FUNCTION_BLOCK Signal EXTENDS InstancePath IMPLEMENTS IBaseSignal, IDifferentiable, ISignal
VAR
    _out : LREAL;
    _derivative : Derivative;
    _iir : InfiniteImpulseResponse;
    _controller : IController;
END_VAR

METHOD Control : IOut
VAR_INPUT
    setpoint : LREAL;
END_VAR
IF _controller <> 0 THEN
    _controller.Update(setpoint:=setpoint, actual:=THIS^.Out);
    _out := _controller.Out;
    Control := THIS^;
ELSE
    ADSLOGSTR(
        msgCtrlMask:=ADSLOG_MSGTYPE_ERROR,
        msgFmtStr:='%s: Assign a controller before calling this method.',
        strArg:=_path
    );
END_IF
END_METHOD

PROPERTY Controller : IController
SET
_controller := Controller;
END_SET
END_PROPERTY

METHOD Differentiate : IDifferentiable
VAR_INPUT
    deltaTime : Millisecond;
END_VAR
_derivative(value:=THIS^.Out, deltaTime:=deltaTime);
_out := _derivative.Out;
Differentiate := THIS^;
END_METHOD

METHOD Iir : IBaseSignal
VAR_INPUT
    decay : LREAL;
END_VAR
_iir(new:=THIS^.Out, decay:=decay);
_out := _iir.Out;
Iir := THIS^;
END_METHOD

PROPERTY Out : LREAL
GET
OUT := _out;
END_GET
END_PROPERTY

METHOD Update : ISignal
VAR_INPUT
    value : LREAL;
END_VAR
_out := value;
Update := THIS^;
END_METHOD

END_FUNCTION_BLOCK

(* stored: Version 1.1.0.1
   POU Signal: Id {d5e65a98-c59a-40a4-8e08-14b2a0104701}, SpecialFunc None
   Method Control: Id {8dcf8e28-9ea3-49a8-b60f-0e1e6205b9e1}
   Property Controller: Id {7fb07e13-2348-48d3-8313-9eff675207f8}
   Set Set: Id {17a680e5-7bae-43e2-91a2-a31ebdb6de08}
   Method Differentiate: Id {3cb626dd-f306-4dd7-8b41-c5d14146e141}
   Method Iir: Id {20733bae-2f54-4e93-a73e-666694dd4f84}
   Property Out: Id {f11c0c9d-cbae-4516-9e11-e42329123126}
   Get Get: Id {42b506ae-6bce-45b3-bdd7-aeb51ebf09f3}
   Method Update: Id {b3adbb0a-1822-4d69-af6d-8f51c8ee0a1c} *)
